FUNCTION_BLOCK SAMPLE_1 (* Single variable sampling *)
  (* Standard: 61499-1; Function: Sampling; Type: Single-variable *)
  (* Version 0.0, 2002-02-15, JHC, Rockwell Automation *)
  (* Compiler header: package fb.rt.math; *)
  (* Compiler Java IBM VisualAge 3.0 *)
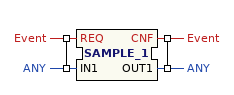
  EVENT_INPUT
    REQ WITH IN1; (* Request to Sample with Monitor Lock *)
  END_EVENT
  EVENT_OUTPUT
    CNF WITH OUT1; (* Initial Sample or OUT1 changed *)
  END_EVENT
  VAR_INPUT
    IN1 : ANY; (* Data to Sample *)
  END_VAR
  VAR_OUTPUT
    OUT1 : ANY; (* Sampled Data *)
  END_VAR
  SERVICE APPLICATION/SAMPLE_1
    SEQUENCE initial_sample_or_data_change
      APPLICATION.REQ(IN1) -> SAMPLE.isDataChanged(IN1,OUT1) -> SAMPLE.copyData(IN1,OUT1) -> APPLICATION.CNF(OUT1);
    END_SEQUENCE
    SEQUENCE no_data_change
      APPLICATION.REQ(IN1) -> SAMPLE.isDataChanged(IN1,OUT1);
    END_SEQUENCE
  END_SERVICE
END_FUNCTION_BLOCK
